// TIA Portal V18 export
ORGANIZATION_BLOCK "11-Bridge Movements"   // OB123, LAD, ProgramCycle
TITLE = Wheel
{ S7_Optimized_Access := 'TRUE' }
VERSION : 0.1
// stored: AutoNumber true, IsIECCheckEnabled false, SetENOAutomatically false
   VAR_INPUT
      Initial_Call : Bool;   // Initial call of this OB
      Remanence : Bool;   // =True, if remanent data are available
   END_VAR
   VAR_TEMP   // added for the SCL form of the ladder/FBD networks
      _w1 : Bool;
      _w2 : Bool;
      _w3 : Bool;
      _w4 : Bool;
   END_VAR
BEGIN

REGION Network 1: JoyStick MID
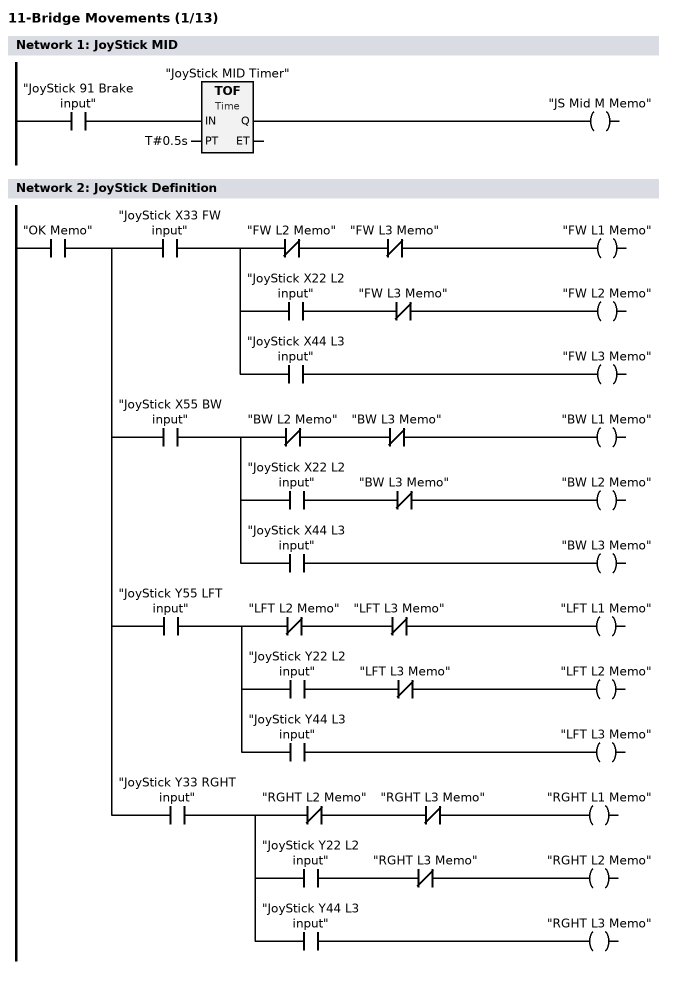
   RUNG wire#powerrail
      Contact( "JoyStick 91 Brake input" )
      { S7_Templates := "time_type := Time" } "JoyStick MID Timer".TOF(pt := T#0.5s, et =>)
      Coil( "JS Mid M Memo" )
   END_RUNG
   // the same network as SCL:
   "JoyStick MID Timer".TOF(IN := "JoyStick 91 Brake input", PT := T#0.5s);
   "JS Mid M Memo" := "JoyStick MID Timer".Q;
END_REGION

REGION Network 2: JoyStick Definition
   RUNG wire#powerrail
      Contact( "OK Memo" )
      wire#w1
      Contact( "JoyStick X33 FW input" )
      wire#w2
      I_Contact( "FW L2 Memo" )
      I_Contact( "FW L3 Memo" )
      Coil( "FW L1 Memo" )
   END_RUNG
   RUNG wire#w2
      Contact( "JoyStick X22 L2 input" )
      I_Contact( "FW L3 Memo" )
      Coil( "FW L2 Memo" )
   END_RUNG
   RUNG wire#w2
      Contact( "JoyStick X44 L3 input" )
      Coil( "FW L3 Memo" )
   END_RUNG
   RUNG wire#w1
      Contact( "JoyStick X55 BW input" )
      wire#w3
      I_Contact( "BW L2 Memo" )
      I_Contact( "BW L3 Memo" )
      Coil( "BW L1 Memo" )
   END_RUNG
   RUNG wire#w3
      Contact( "JoyStick X22 L2 input" )
      I_Contact( "BW L3 Memo" )
      Coil( "BW L2 Memo" )
   END_RUNG
   RUNG wire#w3
      Contact( "JoyStick X44 L3 input" )
      Coil( "BW L3 Memo" )
   END_RUNG
   RUNG wire#w1
      Contact( "JoyStick Y55 LFT input" )
      wire#w4
      I_Contact( "LFT L2 Memo" )
      I_Contact( "LFT L3 Memo" )
      Coil( "LFT L1 Memo" )
   END_RUNG
   RUNG wire#w4
      Contact( "JoyStick Y22 L2 input" )
      I_Contact( "LFT L3 Memo" )
      Coil( "LFT L2 Memo" )
   END_RUNG
   RUNG wire#w4
      Contact( "JoyStick Y44 L3 input" )
      Coil( "LFT L3 Memo" )
   END_RUNG
   RUNG wire#w1
      Contact( "JoyStick Y33 RGHT input" )
      wire#w5
      I_Contact( "RGHT L2 Memo" )
      I_Contact( "RGHT L3 Memo" )
      Coil( "RGHT L1 Memo" )
   END_RUNG
   RUNG wire#w5
      Contact( "JoyStick Y22 L2 input" )
      I_Contact( "RGHT L3 Memo" )
      Coil( "RGHT L2 Memo" )
   END_RUNG
   RUNG wire#w5
      Contact( "JoyStick Y44 L3 input" )
      Coil( "RGHT L3 Memo" )
   END_RUNG
   // the same network as SCL:
   #_w1 := "OK Memo" AND "JoyStick X33 FW input";
   "FW L1 Memo" := #_w1 AND NOT "FW L2 Memo" AND NOT "FW L3 Memo";
   "FW L2 Memo" := #_w1 AND "JoyStick X22 L2 input" AND NOT "FW L3 Memo";
   "FW L3 Memo" := #_w1 AND "JoyStick X44 L3 input";
   #_w2 := "OK Memo" AND "JoyStick X55 BW input";
   "BW L1 Memo" := #_w2 AND NOT "BW L2 Memo" AND NOT "BW L3 Memo";
   "BW L2 Memo" := #_w2 AND "JoyStick X22 L2 input" AND NOT "BW L3 Memo";
   "BW L3 Memo" := #_w2 AND "JoyStick X44 L3 input";
   #_w3 := "OK Memo" AND "JoyStick Y55 LFT input";
   "LFT L1 Memo" := #_w3 AND NOT "LFT L2 Memo" AND NOT "LFT L3 Memo";
   "LFT L2 Memo" := #_w3 AND "JoyStick Y22 L2 input" AND NOT "LFT L3 Memo";
   "LFT L3 Memo" := #_w3 AND "JoyStick Y44 L3 input";
   #_w4 := "OK Memo" AND "JoyStick Y33 RGHT input";
   "RGHT L1 Memo" := #_w4 AND NOT "RGHT L2 Memo" AND NOT "RGHT L3 Memo";
   "RGHT L2 Memo" := #_w4 AND "JoyStick Y22 L2 input" AND NOT "RGHT L3 Memo";
   "RGHT L3 Memo" := #_w4 AND "JoyStick Y44 L3 input";
END_REGION

REGION Network 3: JoyStick Cross Definition
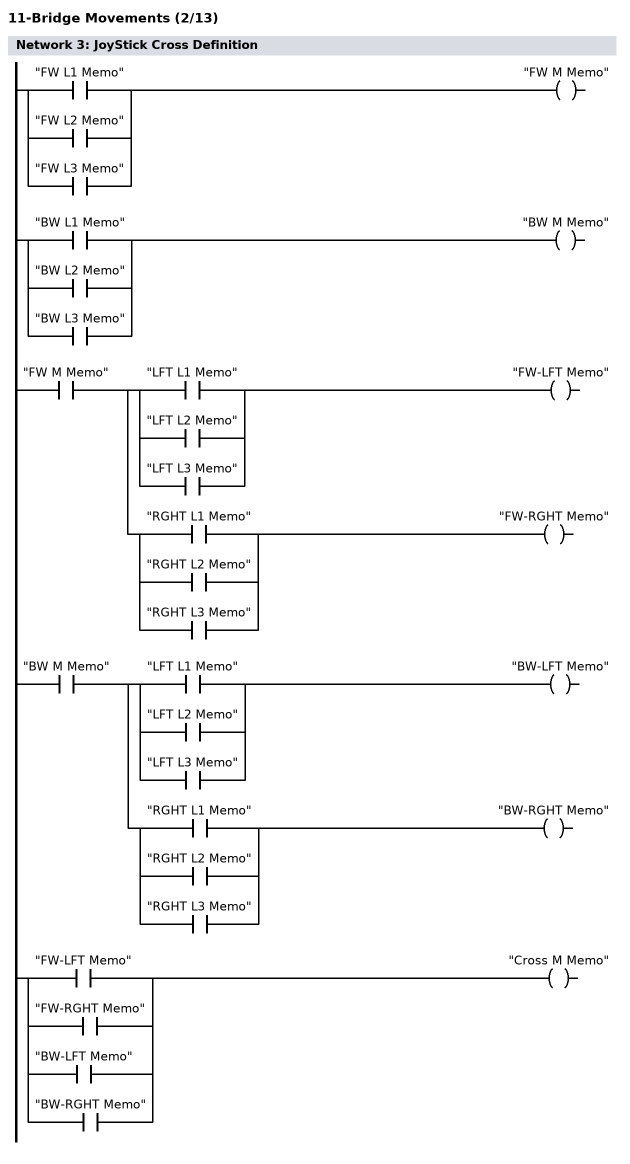
   RUNG wire#powerrail
      Contact( "FW L1 Memo" )
      wire#w1
      Coil( "FW M Memo" )
   END_RUNG
   RUNG wire#powerrail
      Contact( "FW L2 Memo" )
   END_RUNG wire#w1
   RUNG wire#powerrail
      Contact( "FW L3 Memo" )
   END_RUNG wire#w1
   RUNG wire#powerrail
      Contact( "BW L1 Memo" )
      wire#w2
      Coil( "BW M Memo" )
   END_RUNG
   RUNG wire#powerrail
      Contact( "BW L2 Memo" )
   END_RUNG wire#w2
   RUNG wire#powerrail
      Contact( "BW L3 Memo" )
   END_RUNG wire#w2
   RUNG wire#powerrail
      Contact( "FW M Memo" )
      wire#w3
      Contact( "LFT L1 Memo" )
      wire#w4
      Coil( "FW-LFT Memo" )
   END_RUNG
   RUNG wire#w3
      Contact( "LFT L2 Memo" )
   END_RUNG wire#w4
   RUNG wire#w3
      Contact( "LFT L3 Memo" )
   END_RUNG wire#w4
   RUNG wire#w3
      Contact( "RGHT L1 Memo" )
      wire#w5
      Coil( "FW-RGHT Memo" )
   END_RUNG
   RUNG wire#w3
      Contact( "RGHT L2 Memo" )
   END_RUNG wire#w5
   RUNG wire#w3
      Contact( "RGHT L3 Memo" )
   END_RUNG wire#w5
   RUNG wire#powerrail
      Contact( "BW M Memo" )
      wire#w6
      Contact( "LFT L1 Memo" )
      wire#w7
      Coil( "BW-LFT Memo" )
   END_RUNG
   RUNG wire#w6
      Contact( "LFT L2 Memo" )
   END_RUNG wire#w7
   RUNG wire#w6
      Contact( "LFT L3 Memo" )
   END_RUNG wire#w7
   RUNG wire#w6
      Contact( "RGHT L1 Memo" )
      wire#w8
      Coil( "BW-RGHT Memo" )
   END_RUNG
   RUNG wire#w6
      Contact( "RGHT L2 Memo" )
   END_RUNG wire#w8
   RUNG wire#w6
      Contact( "RGHT L3 Memo" )
   END_RUNG wire#w8
   RUNG wire#powerrail
      Contact( "FW-LFT Memo" )
      wire#w9
      Coil( "Cross M Memo" )
   END_RUNG
   RUNG wire#powerrail
      Contact( "FW-RGHT Memo" )
   END_RUNG wire#w9
   RUNG wire#powerrail
      Contact( "BW-LFT Memo" )
   END_RUNG wire#w9
   RUNG wire#powerrail
      Contact( "BW-RGHT Memo" )
   END_RUNG wire#w9
   // the same network as SCL:
   "FW M Memo" := "FW L1 Memo" OR "FW L2 Memo" OR "FW L3 Memo";
   "BW M Memo" := "BW L1 Memo" OR "BW L2 Memo" OR "BW L3 Memo";
   "FW-LFT Memo" := "FW M Memo" AND ("LFT L1 Memo" OR "LFT L2 Memo" OR "LFT L3 Memo");
   "FW-RGHT Memo" := "FW M Memo" AND ("RGHT L1 Memo" OR "RGHT L2 Memo" OR "RGHT L3 Memo");
   "BW-LFT Memo" := "BW M Memo" AND ("LFT L1 Memo" OR "LFT L2 Memo" OR "LFT L3 Memo");
   "BW-RGHT Memo" := "BW M Memo" AND ("RGHT L1 Memo" OR "RGHT L2 Memo" OR "RGHT L3 Memo");
   "Cross M Memo" := "FW-LFT Memo" OR "FW-RGHT Memo" OR "BW-LFT Memo" OR "BW-RGHT Memo";
END_REGION

REGION Network 4: Speed Settings
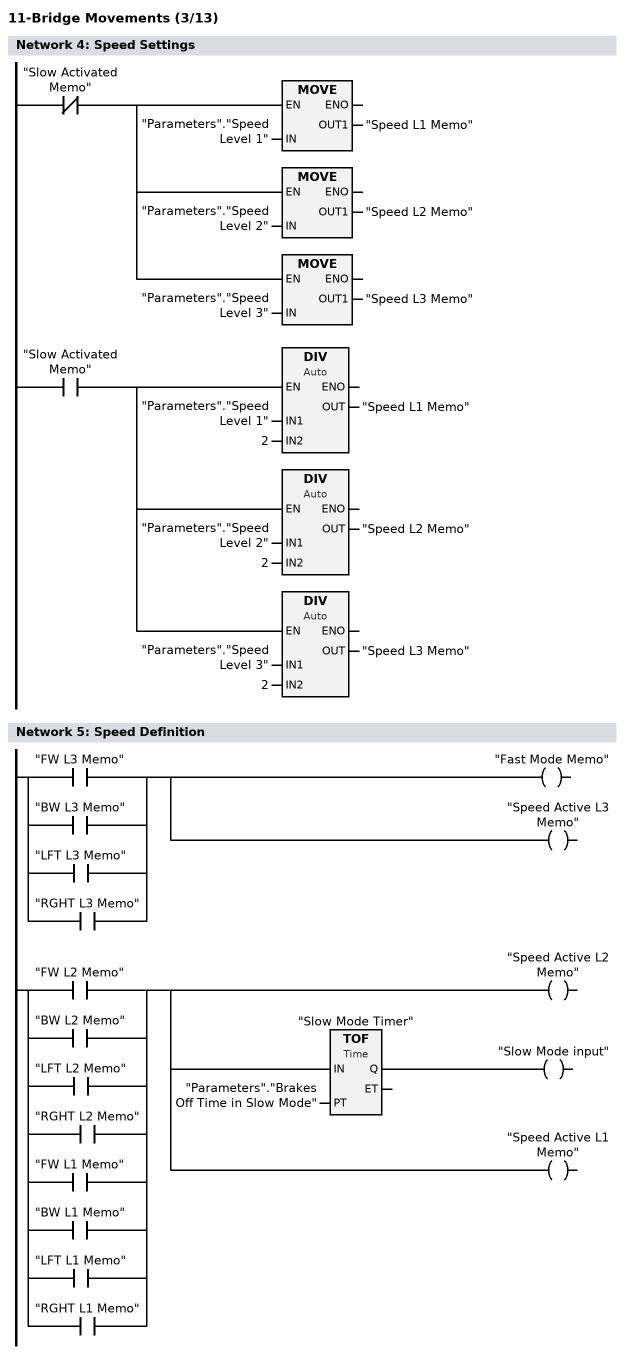
   RUNG wire#powerrail
      I_Contact( "Slow Activated Memo" )
      wire#w1
      Move(in := "Parameters"."Speed Level 1", out1 => "Speed L1 Memo")
   END_RUNG
   RUNG wire#w1
      Move(in := "Parameters"."Speed Level 2", out1 => "Speed L2 Memo")
   END_RUNG
   RUNG wire#w1
      Move(in := "Parameters"."Speed Level 3", out1 => "Speed L3 Memo")
   END_RUNG
   RUNG wire#powerrail
      Contact( "Slow Activated Memo" )
      wire#w2
      Div(in1 := "Parameters"."Speed Level 1", in2 := 2, out => "Speed L1 Memo")
   END_RUNG
   RUNG wire#w2
      Div(in1 := "Parameters"."Speed Level 2", in2 := 2, out => "Speed L2 Memo")
   END_RUNG
   RUNG wire#w2
      Div(in1 := "Parameters"."Speed Level 3", in2 := 2, out => "Speed L3 Memo")
   END_RUNG
   // the same network as SCL:
   IF NOT "Slow Activated Memo" THEN
       "Speed L1 Memo" := "Parameters"."Speed Level 1";
       "Speed L2 Memo" := "Parameters"."Speed Level 2";
       "Speed L3 Memo" := "Parameters"."Speed Level 3";
   END_IF;
   IF "Slow Activated Memo" THEN
       "Speed L1 Memo" := "Parameters"."Speed Level 1" / 2;
       "Speed L2 Memo" := "Parameters"."Speed Level 2" / 2;
       "Speed L3 Memo" := "Parameters"."Speed Level 3" / 2;
   END_IF;
END_REGION

REGION Network 5: Speed Definition
   RUNG wire#powerrail
      Contact( "FW L3 Memo" )
      wire#w1
      Coil( "Fast Mode Memo" )
   END_RUNG
   RUNG wire#powerrail
      Contact( "BW L3 Memo" )
   END_RUNG wire#w1
   RUNG wire#powerrail
      Contact( "LFT L3 Memo" )
   END_RUNG wire#w1
   RUNG wire#powerrail
      Contact( "RGHT L3 Memo" )
   END_RUNG wire#w1
   RUNG wire#w1
      Coil( "Speed Active L3 Memo" )
   END_RUNG
   RUNG wire#powerrail
      Contact( "FW L2 Memo" )
      wire#w2
      Coil( "Speed Active L2 Memo" )
   END_RUNG
   RUNG wire#powerrail
      Contact( "BW L2 Memo" )
   END_RUNG wire#w2
   RUNG wire#powerrail
      Contact( "LFT L2 Memo" )
   END_RUNG wire#w2
   RUNG wire#powerrail
      Contact( "RGHT L2 Memo" )
   END_RUNG wire#w2
   RUNG wire#powerrail
      Contact( "FW L1 Memo" )
   END_RUNG wire#w2
   RUNG wire#powerrail
      Contact( "BW L1 Memo" )
   END_RUNG wire#w2
   RUNG wire#powerrail
      Contact( "LFT L1 Memo" )
   END_RUNG wire#w2
   RUNG wire#powerrail
      Contact( "RGHT L1 Memo" )
   END_RUNG wire#w2
   RUNG wire#w2
      { S7_Templates := "time_type := Time" } "Slow Mode Timer".TOF(pt := "Parameters"."Brakes Off Time in Slow Mode", et =>)
      Coil( "Slow Mode input" )
   END_RUNG
   RUNG wire#w2
      Coil( "Speed Active L1 Memo" )
   END_RUNG
   // the same network as SCL:
   "Fast Mode Memo" := "FW L3 Memo" OR "BW L3 Memo" OR "LFT L3 Memo" OR "RGHT L3 Memo";
   "Speed Active L3 Memo" := "Fast Mode Memo";
   "Speed Active L2 Memo" := "FW L2 Memo" OR "BW L2 Memo" OR "LFT L2 Memo" OR "RGHT L2 Memo" OR "FW L1 Memo" OR "BW L1 Memo" OR "LFT L1 Memo" OR "RGHT L1 Memo";
   "Slow Mode Timer".TOF(IN := "Speed Active L2 Memo", PT := "Parameters"."Brakes Off Time in Slow Mode");
   "Slow Mode input" := "Slow Mode Timer".Q;
   "Speed Active L1 Memo" := "Speed Active L2 Memo";
END_REGION

REGION Network 6: Slow Activated
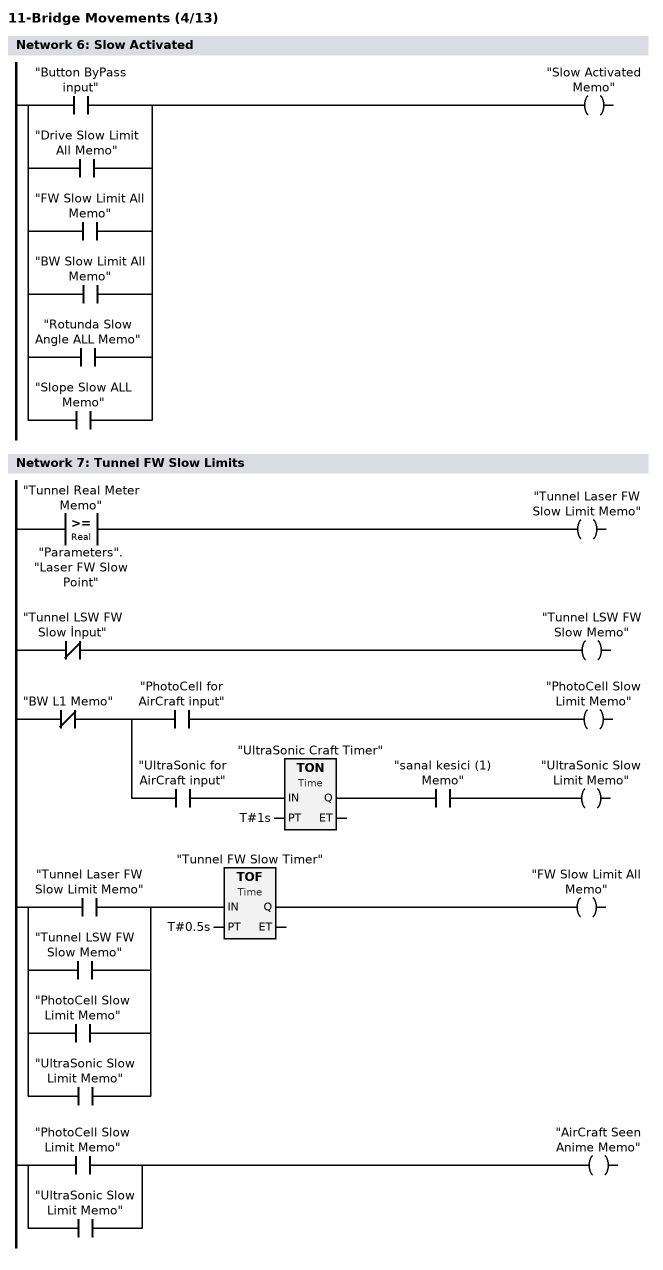
   RUNG wire#powerrail
      Contact( "Button ByPass input" )
      wire#w1
      Coil( "Slow Activated Memo" )
   END_RUNG
   RUNG wire#powerrail
      Contact( "Drive Slow Limit All Memo" )
   END_RUNG wire#w1
   RUNG wire#powerrail
      Contact( "FW Slow Limit All Memo" )
   END_RUNG wire#w1
   RUNG wire#powerrail
      Contact( "BW Slow Limit All Memo" )
   END_RUNG wire#w1
   RUNG wire#powerrail
      Contact( "Rotunda Slow Angle ALL Memo" )
   END_RUNG wire#w1
   RUNG wire#powerrail
      Contact( "Slope Slow ALL Memo" )
   END_RUNG wire#w1
   // the same network as SCL:
   "Slow Activated Memo" := "Button ByPass input" OR "Drive Slow Limit All Memo" OR "FW Slow Limit All Memo" OR "BW Slow Limit All Memo" OR "Rotunda Slow Angle ALL Memo" OR "Slope Slow ALL Memo";
END_REGION

REGION Network 7: Tunnel FW Slow Limits
   RUNG wire#powerrail
      { S7_Templates := "SrcType := Real" } GE_Contact(in1 := "Tunnel Real Meter Memo", in2 := "Parameters"."Laser FW Slow Point")
      Coil( "Tunnel Laser FW Slow Limit Memo" )
   END_RUNG
   RUNG wire#powerrail
      I_Contact( "Tunnel LSW FW Slow İnput" )
      Coil( "Tunnel LSW FW Slow Memo" )
   END_RUNG
   RUNG wire#powerrail
      I_Contact( "BW L1 Memo" )
      wire#w1
      Contact( "PhotoCell for AirCraft input" )
      Coil( "PhotoCell Slow Limit Memo" )
   END_RUNG
   RUNG wire#w1
      Contact( "UltraSonic for AirCraft input" )
      { S7_Templates := "time_type := Time" } "UltraSonic Craft Timer".TON(pt := T#1s, et =>)
      Contact( "sanal kesici (1) Memo" )
      Coil( "UltraSonic Slow Limit Memo" )
   END_RUNG
   RUNG wire#powerrail
      Contact( "Tunnel Laser FW Slow Limit Memo" )
      wire#w2
      { S7_Templates := "time_type := Time" } "Tunnel FW Slow Timer".TOF(pt := T#0.5s, et =>)
      Coil( "FW Slow Limit All Memo" )
   END_RUNG
   RUNG wire#powerrail
      Contact( "Tunnel LSW FW Slow Memo" )
   END_RUNG wire#w2
   RUNG wire#powerrail
      Contact( "PhotoCell Slow Limit Memo" )
   END_RUNG wire#w2
   RUNG wire#powerrail
      Contact( "UltraSonic Slow Limit Memo" )
   END_RUNG wire#w2
   RUNG wire#powerrail
      Contact( "PhotoCell Slow Limit Memo" )
      wire#w3
      Coil( "AirCraft Seen Anime Memo" )
   END_RUNG
   RUNG wire#powerrail
      Contact( "UltraSonic Slow Limit Memo" )
   END_RUNG wire#w3
   // the same network as SCL:
   "Tunnel Laser FW Slow Limit Memo" := "Tunnel Real Meter Memo" >= "Parameters"."Laser FW Slow Point";
   "Tunnel LSW FW Slow Memo" := NOT "Tunnel LSW FW Slow İnput";
   "PhotoCell Slow Limit Memo" := NOT "BW L1 Memo" AND "PhotoCell for AirCraft input";
   "UltraSonic Craft Timer".TON(IN := NOT "BW L1 Memo" AND "UltraSonic for AirCraft input", PT := T#1s);
   "UltraSonic Slow Limit Memo" := "UltraSonic Craft Timer".Q AND "sanal kesici (1) Memo";
   "Tunnel FW Slow Timer".TOF(IN := "Tunnel Laser FW Slow Limit Memo" OR "Tunnel LSW FW Slow Memo" OR "PhotoCell Slow Limit Memo" OR "UltraSonic Slow Limit Memo",
                           PT := T#0.5s);
   "FW Slow Limit All Memo" := "Tunnel FW Slow Timer".Q;
   "AirCraft Seen Anime Memo" := "PhotoCell Slow Limit Memo" OR "UltraSonic Slow Limit Memo";
END_REGION

REGION Network 8: Tunnel BW Slow Limits
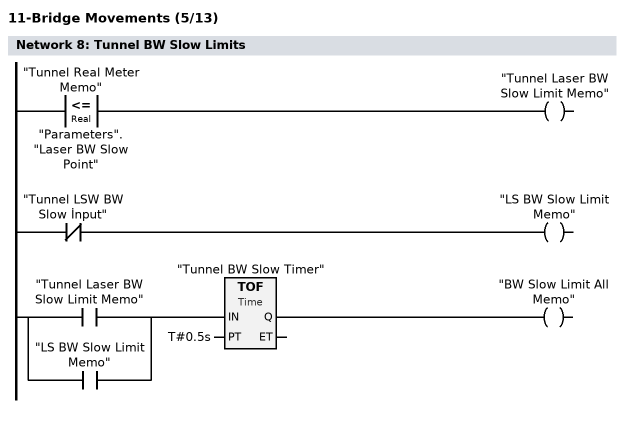
   RUNG wire#powerrail
      { S7_Templates := "SrcType := Real" } LE_Contact(in1 := "Tunnel Real Meter Memo", in2 := "Parameters"."Laser BW Slow Point")
      Coil( "Tunnel Laser BW Slow Limit Memo" )
   END_RUNG
   RUNG wire#powerrail
      I_Contact( "Tunnel LSW BW Slow İnput" )
      Coil( "LS BW Slow Limit Memo" )
   END_RUNG
   RUNG wire#powerrail
      Contact( "Tunnel Laser BW Slow Limit Memo" )
      wire#w1
      { S7_Templates := "time_type := Time" } "Tunnel BW Slow Timer".TOF(pt := T#0.5s, et =>)
      Coil( "BW Slow Limit All Memo" )
   END_RUNG
   RUNG wire#powerrail
      Contact( "LS BW Slow Limit Memo" )
   END_RUNG wire#w1
   // the same network as SCL:
   "Tunnel Laser BW Slow Limit Memo" := "Tunnel Real Meter Memo" <= "Parameters"."Laser BW Slow Point";
   "LS BW Slow Limit Memo" := NOT "Tunnel LSW BW Slow İnput";
   "Tunnel BW Slow Timer".TOF(IN := "Tunnel Laser BW Slow Limit Memo" OR "LS BW Slow Limit Memo", PT := T#0.5s);
   "BW Slow Limit All Memo" := "Tunnel BW Slow Timer".Q;
END_REGION

REGION Network 9: Tunnel FW Stop Limits
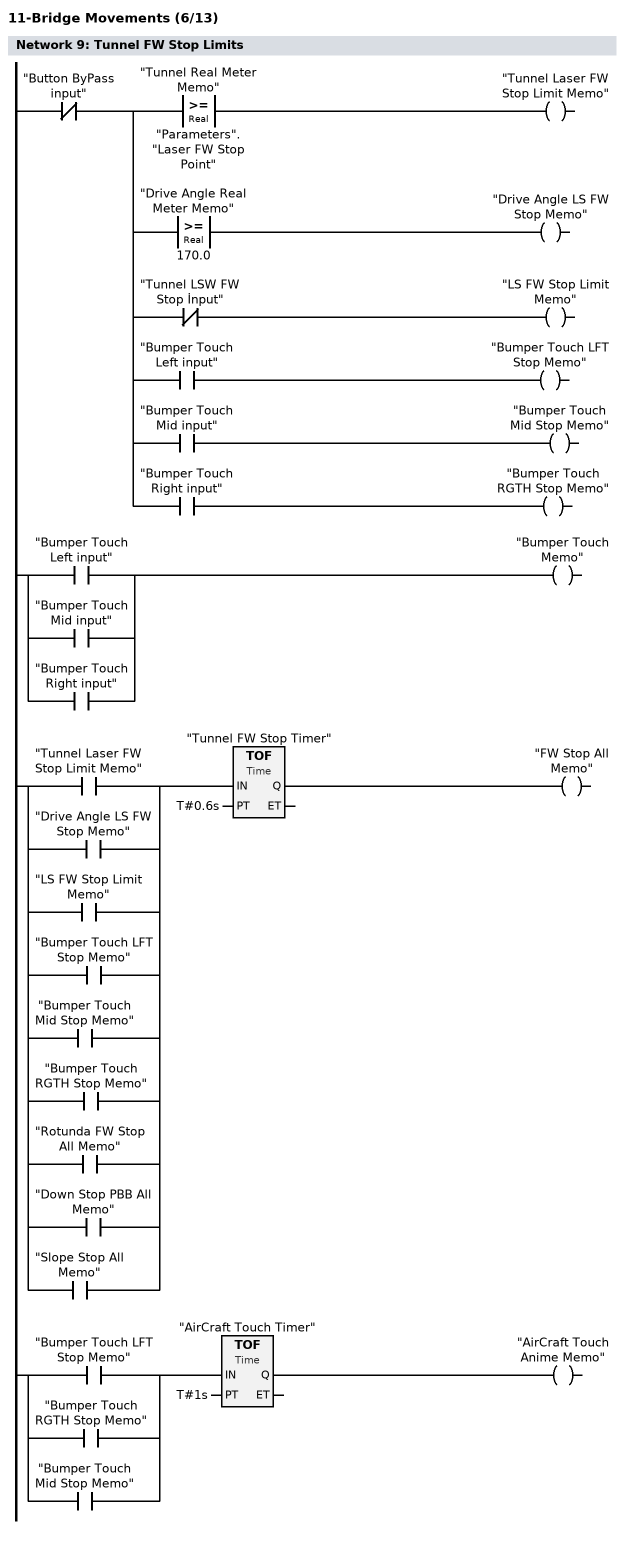
   RUNG wire#powerrail
      I_Contact( "Button ByPass input" )
      wire#w1
      { S7_Templates := "SrcType := Real" } GE_Contact(in1 := "Tunnel Real Meter Memo", in2 := "Parameters"."Laser FW Stop Point")
      Coil( "Tunnel Laser FW Stop Limit Memo" )
   END_RUNG
   RUNG wire#w1
      { S7_Templates := "SrcType := Real" } GE_Contact(in1 := "Drive Angle Real Meter Memo", in2 := 170.0)
      Coil( "Drive Angle LS FW Stop Memo" )
   END_RUNG
   RUNG wire#w1
      I_Contact( "Tunnel LSW FW Stop İnput" )
      Coil( "LS FW Stop Limit Memo" )
   END_RUNG
   RUNG wire#w1
      Contact( "Bumper Touch Left input" )
      Coil( "Bumper Touch LFT Stop Memo" )
   END_RUNG
   RUNG wire#w1
      Contact( "Bumper Touch Mid input" )
      Coil( "Bumper Touch Mid Stop Memo" )
   END_RUNG
   RUNG wire#w1
      Contact( "Bumper Touch Right input" )
      Coil( "Bumper Touch RGTH Stop Memo" )
   END_RUNG
   RUNG wire#powerrail
      Contact( "Bumper Touch Left input" )
      wire#w2
      Coil( "Bumper Touch Memo" )
   END_RUNG
   RUNG wire#powerrail
      Contact( "Bumper Touch Mid input" )
   END_RUNG wire#w2
   RUNG wire#powerrail
      Contact( "Bumper Touch Right input" )
   END_RUNG wire#w2
   RUNG wire#powerrail
      Contact( "Tunnel Laser FW Stop Limit Memo" )
      wire#w3
      { S7_Templates := "time_type := Time" } "Tunnel FW Stop Timer".TOF(pt := T#0.6s, et =>)
      Coil( "FW Stop All Memo" )
   END_RUNG
   RUNG wire#powerrail
      Contact( "Drive Angle LS FW Stop Memo" )
   END_RUNG wire#w3
   RUNG wire#powerrail
      Contact( "LS FW Stop Limit Memo" )
   END_RUNG wire#w3
   RUNG wire#powerrail
      Contact( "Bumper Touch LFT Stop Memo" )
   END_RUNG wire#w3
   RUNG wire#powerrail
      Contact( "Bumper Touch Mid Stop Memo" )
   END_RUNG wire#w3
   RUNG wire#powerrail
      Contact( "Bumper Touch RGTH Stop Memo" )
   END_RUNG wire#w3
   RUNG wire#powerrail
      Contact( "Rotunda FW Stop All Memo" )
   END_RUNG wire#w3
   RUNG wire#powerrail
      Contact( "Down Stop PBB All Memo" )
   END_RUNG wire#w3
   RUNG wire#powerrail
      Contact( "Slope Stop All Memo" )
   END_RUNG wire#w3
   RUNG wire#powerrail
      Contact( "Bumper Touch LFT Stop Memo" )
      wire#w4
      { S7_Templates := "time_type := Time" } "AirCraft Touch Timer".TOF(pt := T#1s, et =>)
      Coil( "AirCraft Touch Anime Memo" )
   END_RUNG
   RUNG wire#powerrail
      Contact( "Bumper Touch RGTH Stop Memo" )
   END_RUNG wire#w4
   RUNG wire#powerrail
      Contact( "Bumper Touch Mid Stop Memo" )
   END_RUNG wire#w4
   // the same network as SCL:
   #_w1 := NOT "Button ByPass input";
   "Tunnel Laser FW Stop Limit Memo" := #_w1 AND ("Tunnel Real Meter Memo" >= "Parameters"."Laser FW Stop Point");
   "Drive Angle LS FW Stop Memo" := #_w1 AND ("Drive Angle Real Meter Memo" >= 170.0);
   "LS FW Stop Limit Memo" := #_w1 AND NOT "Tunnel LSW FW Stop İnput";
   "Bumper Touch LFT Stop Memo" := #_w1 AND "Bumper Touch Left input";
   "Bumper Touch Mid Stop Memo" := #_w1 AND "Bumper Touch Mid input";
   "Bumper Touch RGTH Stop Memo" := #_w1 AND "Bumper Touch Right input";
   "Bumper Touch Memo" := "Bumper Touch Left input" OR "Bumper Touch Mid input" OR "Bumper Touch Right input";
   "Tunnel FW Stop Timer".TOF(IN := "Tunnel Laser FW Stop Limit Memo" OR "Drive Angle LS FW Stop Memo" OR "LS FW Stop Limit Memo" OR "Bumper Touch LFT Stop Memo" OR "Bumper Touch Mid Stop Memo" OR "Bumper Touch RGTH Stop Memo" OR "Rotunda FW Stop All Memo" OR "Down Stop PBB All Memo" OR "Slope Stop All Memo",
                           PT := T#0.6s);
   "FW Stop All Memo" := "Tunnel FW Stop Timer".Q;
   "AirCraft Touch Timer".TOF(IN := "Bumper Touch LFT Stop Memo" OR "Bumper Touch RGTH Stop Memo" OR "Bumper Touch Mid Stop Memo",
                           PT := T#1s);
   "AirCraft Touch Anime Memo" := "AirCraft Touch Timer".Q;
END_REGION

REGION Network 10: Tunnel BW Stop Limits
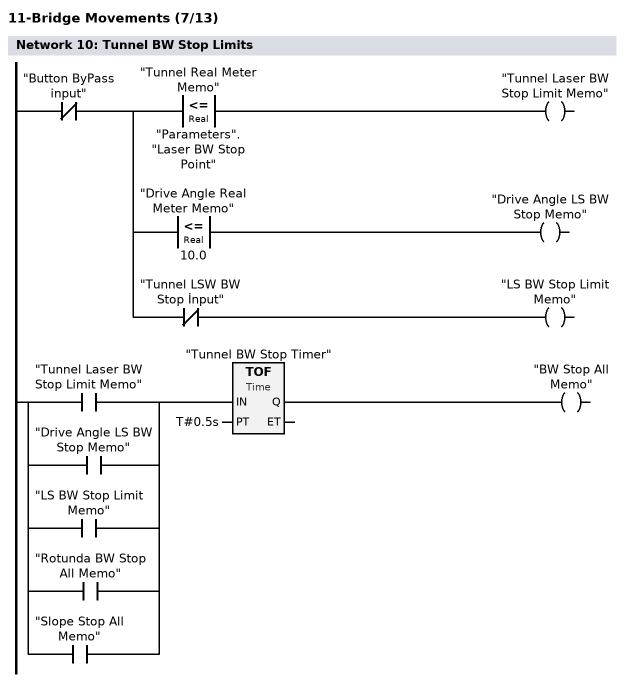
   RUNG wire#powerrail
      I_Contact( "Button ByPass input" )
      wire#w1
      { S7_Templates := "SrcType := Real" } LE_Contact(in1 := "Tunnel Real Meter Memo", in2 := "Parameters"."Laser BW Stop Point")
      Coil( "Tunnel Laser BW Stop Limit Memo" )
   END_RUNG
   RUNG wire#w1
      { S7_Templates := "SrcType := Real" } LE_Contact(in1 := "Drive Angle Real Meter Memo", in2 := 10.0)
      Coil( "Drive Angle LS BW Stop Memo" )
   END_RUNG
   RUNG wire#w1
      I_Contact( "Tunnel LSW BW Stop İnput" )
      Coil( "LS BW Stop Limit Memo" )
   END_RUNG
   RUNG wire#powerrail
      Contact( "Tunnel Laser BW Stop Limit Memo" )
      wire#w2
      { S7_Templates := "time_type := Time" } "Tunnel BW Stop Timer".TOF(pt := T#0.5s, et =>)
      Coil( "BW Stop All Memo" )
   END_RUNG
   RUNG wire#powerrail
      Contact( "Drive Angle LS BW Stop Memo" )
   END_RUNG wire#w2
   RUNG wire#powerrail
      Contact( "LS BW Stop Limit Memo" )
   END_RUNG wire#w2
   RUNG wire#powerrail
      Contact( "Rotunda BW Stop All Memo" )
   END_RUNG wire#w2
   RUNG wire#powerrail
      Contact( "Slope Stop All Memo" )
   END_RUNG wire#w2
   // the same network as SCL:
   #_w1 := NOT "Button ByPass input";
   "Tunnel Laser BW Stop Limit Memo" := #_w1 AND ("Tunnel Real Meter Memo" <= "Parameters"."Laser BW Stop Point");
   "Drive Angle LS BW Stop Memo" := #_w1 AND ("Drive Angle Real Meter Memo" <= 10.0);
   "LS BW Stop Limit Memo" := #_w1 AND NOT "Tunnel LSW BW Stop İnput";
   "Tunnel BW Stop Timer".TOF(IN := "Tunnel Laser BW Stop Limit Memo" OR "Drive Angle LS BW Stop Memo" OR "LS BW Stop Limit Memo" OR "Rotunda BW Stop All Memo" OR "Slope Stop All Memo",
                           PT := T#0.5s);
   "BW Stop All Memo" := "Tunnel BW Stop Timer".Q;
END_REGION

REGION Network 11: Tunnel FW
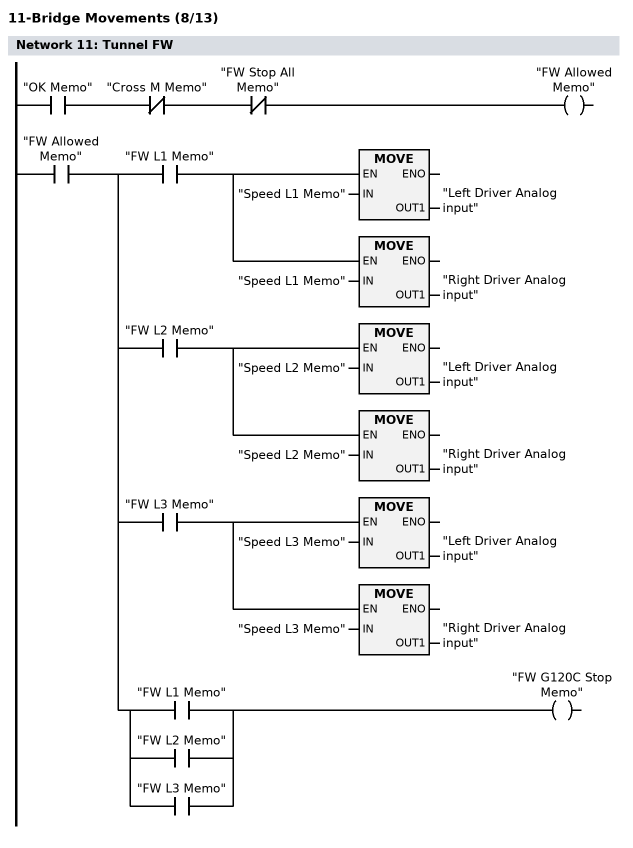
   RUNG wire#powerrail
      Contact( "OK Memo" )
      I_Contact( "Cross M Memo" )
      I_Contact( "FW Stop All Memo" )
      Coil( "FW Allowed Memo" )
   END_RUNG
   RUNG wire#powerrail
      Contact( "FW Allowed Memo" )
      wire#w1
      Contact( "FW L1 Memo" )
      wire#w2
      Move(in := "Speed L1 Memo", out1 => "Left Driver Analog input")
   END_RUNG
   RUNG wire#w2
      Move(in := "Speed L1 Memo", out1 => "Right Driver Analog input")
   END_RUNG
   RUNG wire#w1
      Contact( "FW L2 Memo" )
      wire#w3
      Move(in := "Speed L2 Memo", out1 => "Left Driver Analog input")
   END_RUNG
   RUNG wire#w3
      Move(in := "Speed L2 Memo", out1 => "Right Driver Analog input")
   END_RUNG
   RUNG wire#w1
      Contact( "FW L3 Memo" )
      wire#w4
      Move(in := "Speed L3 Memo", out1 => "Left Driver Analog input")
   END_RUNG
   RUNG wire#w4
      Move(in := "Speed L3 Memo", out1 => "Right Driver Analog input")
   END_RUNG
   RUNG wire#w1
      Contact( "FW L1 Memo" )
      wire#w5
      Coil( "FW G120C Stop Memo" )
   END_RUNG
   RUNG wire#w1
      Contact( "FW L2 Memo" )
   END_RUNG wire#w5
   RUNG wire#w1
      Contact( "FW L3 Memo" )
   END_RUNG wire#w5
   // the same network as SCL:
   "FW Allowed Memo" := "OK Memo" AND NOT "Cross M Memo" AND NOT "FW Stop All Memo";
   IF "FW Allowed Memo" AND "FW L1 Memo" THEN
       "Left Driver Analog input" := "Speed L1 Memo";
       "Right Driver Analog input" := "Speed L1 Memo";
   END_IF;
   IF "FW Allowed Memo" AND "FW L2 Memo" THEN
       "Left Driver Analog input" := "Speed L2 Memo";
       "Right Driver Analog input" := "Speed L2 Memo";
   END_IF;
   IF "FW Allowed Memo" AND "FW L3 Memo" THEN
       "Left Driver Analog input" := "Speed L3 Memo";
       "Right Driver Analog input" := "Speed L3 Memo";
   END_IF;
   "FW G120C Stop Memo" := "FW Allowed Memo" AND ("FW L1 Memo" OR "FW L2 Memo" OR "FW L3 Memo");
END_REGION

REGION Network 12: Tunnel BW
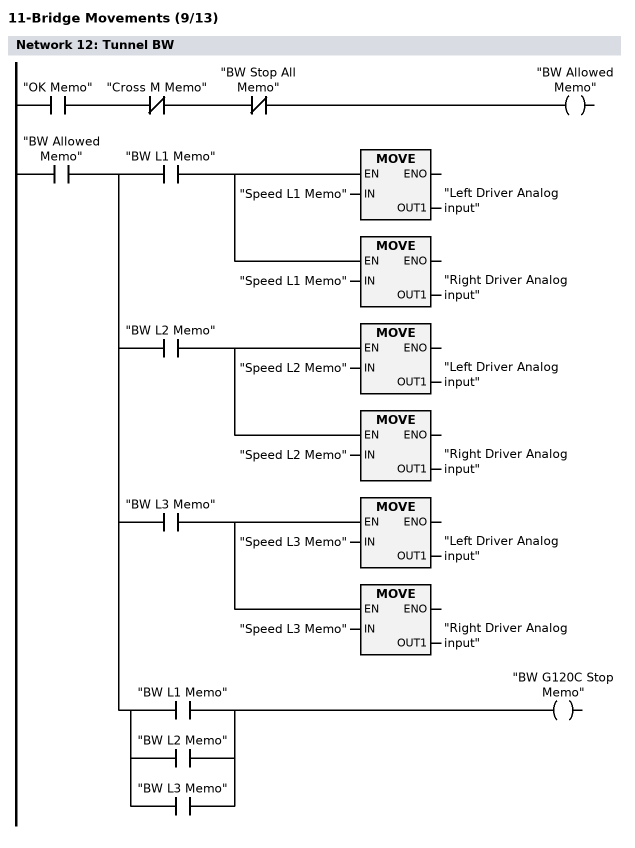
   RUNG wire#powerrail
      Contact( "OK Memo" )
      I_Contact( "Cross M Memo" )
      I_Contact( "BW Stop All Memo" )
      Coil( "BW Allowed Memo" )
   END_RUNG
   RUNG wire#powerrail
      Contact( "BW Allowed Memo" )
      wire#w1
      Contact( "BW L1 Memo" )
      wire#w2
      Move(in := "Speed L1 Memo", out1 => "Left Driver Analog input")
   END_RUNG
   RUNG wire#w2
      Move(in := "Speed L1 Memo", out1 => "Right Driver Analog input")
   END_RUNG
   RUNG wire#w1
      Contact( "BW L2 Memo" )
      wire#w3
      Move(in := "Speed L2 Memo", out1 => "Left Driver Analog input")
   END_RUNG
   RUNG wire#w3
      Move(in := "Speed L2 Memo", out1 => "Right Driver Analog input")
   END_RUNG
   RUNG wire#w1
      Contact( "BW L3 Memo" )
      wire#w4
      Move(in := "Speed L3 Memo", out1 => "Left Driver Analog input")
   END_RUNG
   RUNG wire#w4
      Move(in := "Speed L3 Memo", out1 => "Right Driver Analog input")
   END_RUNG
   RUNG wire#w1
      Contact( "BW L1 Memo" )
      wire#w5
      Coil( "BW G120C Stop Memo" )
   END_RUNG
   RUNG wire#w1
      Contact( "BW L2 Memo" )
   END_RUNG wire#w5
   RUNG wire#w1
      Contact( "BW L3 Memo" )
   END_RUNG wire#w5
   // the same network as SCL:
   "BW Allowed Memo" := "OK Memo" AND NOT "Cross M Memo" AND NOT "BW Stop All Memo";
   IF "BW Allowed Memo" AND "BW L1 Memo" THEN
       "Left Driver Analog input" := "Speed L1 Memo";
       "Right Driver Analog input" := "Speed L1 Memo";
   END_IF;
   IF "BW Allowed Memo" AND "BW L2 Memo" THEN
       "Left Driver Analog input" := "Speed L2 Memo";
       "Right Driver Analog input" := "Speed L2 Memo";
   END_IF;
   IF "BW Allowed Memo" AND "BW L3 Memo" THEN
       "Left Driver Analog input" := "Speed L3 Memo";
       "Right Driver Analog input" := "Speed L3 Memo";
   END_IF;
   "BW G120C Stop Memo" := "BW Allowed Memo" AND ("BW L1 Memo" OR "BW L2 Memo" OR "BW L3 Memo");
END_REGION

REGION Network 13: Tunnel LFT
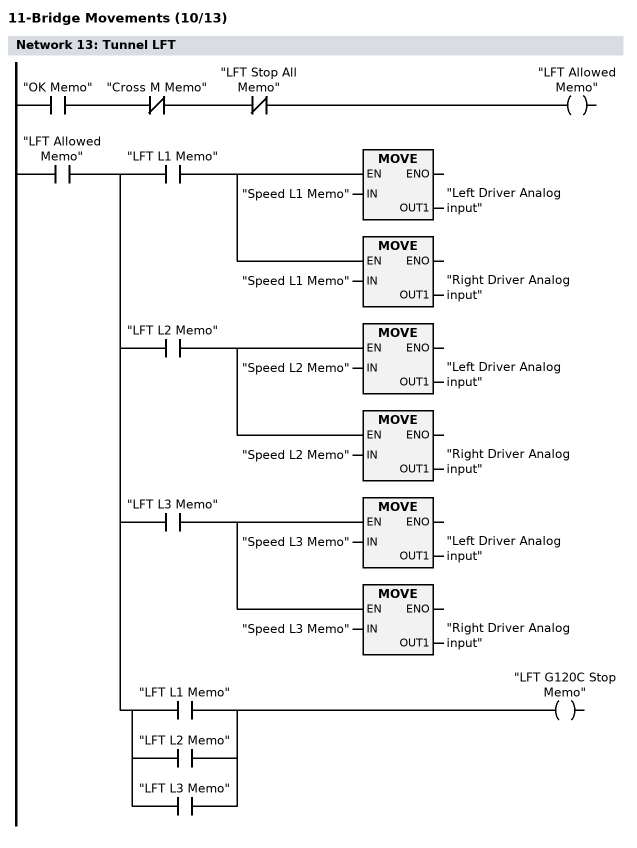
   RUNG wire#powerrail
      Contact( "OK Memo" )
      I_Contact( "Cross M Memo" )
      I_Contact( "LFT Stop All Memo" )
      Coil( "LFT Allowed Memo" )
   END_RUNG
   RUNG wire#powerrail
      Contact( "LFT Allowed Memo" )
      wire#w1
      Contact( "LFT L1 Memo" )
      wire#w2
      Move(in := "Speed L1 Memo", out1 => "Left Driver Analog input")
   END_RUNG
   RUNG wire#w2
      Move(in := "Speed L1 Memo", out1 => "Right Driver Analog input")
   END_RUNG
   RUNG wire#w1
      Contact( "LFT L2 Memo" )
      wire#w3
      Move(in := "Speed L2 Memo", out1 => "Left Driver Analog input")
   END_RUNG
   RUNG wire#w3
      Move(in := "Speed L2 Memo", out1 => "Right Driver Analog input")
   END_RUNG
   RUNG wire#w1
      Contact( "LFT L3 Memo" )
      wire#w4
      Move(in := "Speed L3 Memo", out1 => "Left Driver Analog input")
   END_RUNG
   RUNG wire#w4
      Move(in := "Speed L3 Memo", out1 => "Right Driver Analog input")
   END_RUNG
   RUNG wire#w1
      Contact( "LFT L1 Memo" )
      wire#w5
      Coil( "LFT G120C Stop Memo" )
   END_RUNG
   RUNG wire#w1
      Contact( "LFT L2 Memo" )
   END_RUNG wire#w5
   RUNG wire#w1
      Contact( "LFT L3 Memo" )
   END_RUNG wire#w5
   // the same network as SCL:
   "LFT Allowed Memo" := "OK Memo" AND NOT "Cross M Memo" AND NOT "LFT Stop All Memo";
   IF "LFT Allowed Memo" AND "LFT L1 Memo" THEN
       "Left Driver Analog input" := "Speed L1 Memo";
       "Right Driver Analog input" := "Speed L1 Memo";
   END_IF;
   IF "LFT Allowed Memo" AND "LFT L2 Memo" THEN
       "Left Driver Analog input" := "Speed L2 Memo";
       "Right Driver Analog input" := "Speed L2 Memo";
   END_IF;
   IF "LFT Allowed Memo" AND "LFT L3 Memo" THEN
       "Left Driver Analog input" := "Speed L3 Memo";
       "Right Driver Analog input" := "Speed L3 Memo";
   END_IF;
   "LFT G120C Stop Memo" := "LFT Allowed Memo" AND ("LFT L1 Memo" OR "LFT L2 Memo" OR "LFT L3 Memo");
END_REGION

REGION Network 14: Tunnel RGHT
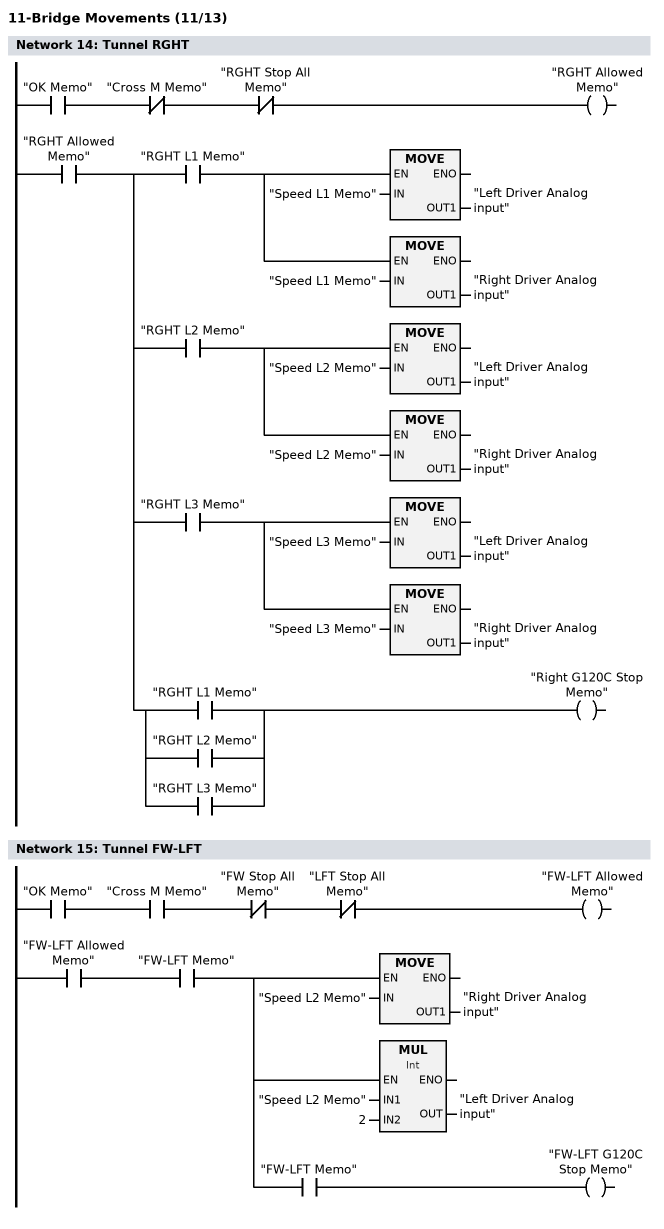
   RUNG wire#powerrail
      Contact( "OK Memo" )
      I_Contact( "Cross M Memo" )
      I_Contact( "RGHT Stop All Memo" )
      Coil( "RGHT Allowed Memo" )
   END_RUNG
   RUNG wire#powerrail
      Contact( "RGHT Allowed Memo" )
      wire#w1
      Contact( "RGHT L1 Memo" )
      wire#w2
      Move(in := "Speed L1 Memo", out1 => "Left Driver Analog input")
   END_RUNG
   RUNG wire#w2
      Move(in := "Speed L1 Memo", out1 => "Right Driver Analog input")
   END_RUNG
   RUNG wire#w1
      Contact( "RGHT L2 Memo" )
      wire#w3
      Move(in := "Speed L2 Memo", out1 => "Left Driver Analog input")
   END_RUNG
   RUNG wire#w3
      Move(in := "Speed L2 Memo", out1 => "Right Driver Analog input")
   END_RUNG
   RUNG wire#w1
      Contact( "RGHT L3 Memo" )
      wire#w4
      Move(in := "Speed L3 Memo", out1 => "Left Driver Analog input")
   END_RUNG
   RUNG wire#w4
      Move(in := "Speed L3 Memo", out1 => "Right Driver Analog input")
   END_RUNG
   RUNG wire#w1
      Contact( "RGHT L1 Memo" )
      wire#w5
      Coil( "Right G120C Stop Memo" )
   END_RUNG
   RUNG wire#w1
      Contact( "RGHT L2 Memo" )
   END_RUNG wire#w5
   RUNG wire#w1
      Contact( "RGHT L3 Memo" )
   END_RUNG wire#w5
   // the same network as SCL:
   "RGHT Allowed Memo" := "OK Memo" AND NOT "Cross M Memo" AND NOT "RGHT Stop All Memo";
   IF "RGHT Allowed Memo" AND "RGHT L1 Memo" THEN
       "Left Driver Analog input" := "Speed L1 Memo";
       "Right Driver Analog input" := "Speed L1 Memo";
   END_IF;
   IF "RGHT Allowed Memo" AND "RGHT L2 Memo" THEN
       "Left Driver Analog input" := "Speed L2 Memo";
       "Right Driver Analog input" := "Speed L2 Memo";
   END_IF;
   IF "RGHT Allowed Memo" AND "RGHT L3 Memo" THEN
       "Left Driver Analog input" := "Speed L3 Memo";
       "Right Driver Analog input" := "Speed L3 Memo";
   END_IF;
   "Right G120C Stop Memo" := "RGHT Allowed Memo" AND ("RGHT L1 Memo" OR "RGHT L2 Memo" OR "RGHT L3 Memo");
END_REGION

REGION Network 15: Tunnel FW-LFT
   RUNG wire#powerrail
      Contact( "OK Memo" )
      Contact( "Cross M Memo" )
      I_Contact( "FW Stop All Memo" )
      I_Contact( "LFT Stop All Memo" )
      Coil( "FW-LFT Allowed Memo" )
   END_RUNG
   RUNG wire#powerrail
      Contact( "FW-LFT Allowed Memo" )
      Contact( "FW-LFT Memo" )
      wire#w1
      Move(in := "Speed L2 Memo", out1 => "Right Driver Analog input")
   END_RUNG
   RUNG wire#w1
      { S7_Templates := "SrcType := Int" } Mul(in1 := "Speed L2 Memo", in2 := 2, out => "Left Driver Analog input")
   END_RUNG
   RUNG wire#w1
      Contact( "FW-LFT Memo" )
      Coil( "FW-LFT G120C Stop Memo" )
   END_RUNG
   // the same network as SCL:
   "FW-LFT Allowed Memo" := "OK Memo" AND "Cross M Memo" AND NOT "FW Stop All Memo" AND NOT "LFT Stop All Memo";
   #_w1 := "FW-LFT Allowed Memo" AND "FW-LFT Memo";
   IF #_w1 THEN
       "Right Driver Analog input" := "Speed L2 Memo";
       "Left Driver Analog input" := "Speed L2 Memo" * 2;
   END_IF;
   "FW-LFT G120C Stop Memo" := #_w1 AND "FW-LFT Memo";
END_REGION

REGION Network 16: Tunnel FW-RGHT
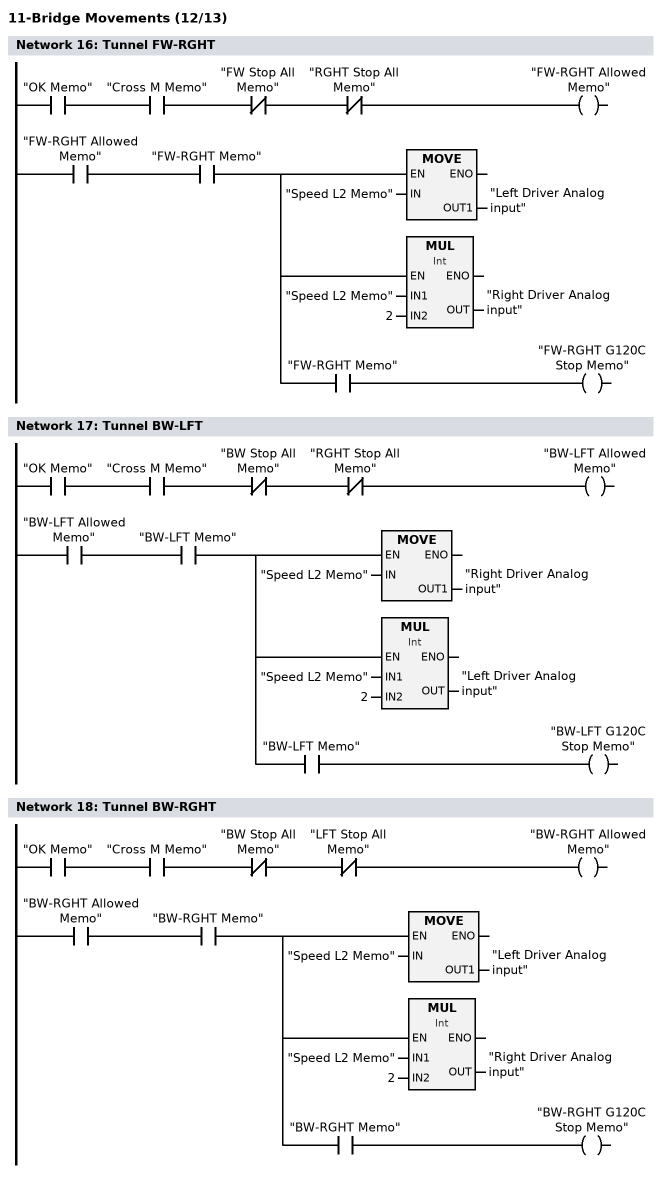
   RUNG wire#powerrail
      Contact( "OK Memo" )
      Contact( "Cross M Memo" )
      I_Contact( "FW Stop All Memo" )
      I_Contact( "RGHT Stop All Memo" )
      Coil( "FW-RGHT Allowed Memo" )
   END_RUNG
   RUNG wire#powerrail
      Contact( "FW-RGHT Allowed Memo" )
      Contact( "FW-RGHT Memo" )
      wire#w1
      Move(in := "Speed L2 Memo", out1 => "Left Driver Analog input")
   END_RUNG
   RUNG wire#w1
      { S7_Templates := "SrcType := Int" } Mul(in1 := "Speed L2 Memo", in2 := 2, out => "Right Driver Analog input")
   END_RUNG
   RUNG wire#w1
      Contact( "FW-RGHT Memo" )
      Coil( "FW-RGHT G120C Stop Memo" )
   END_RUNG
   // the same network as SCL:
   "FW-RGHT Allowed Memo" := "OK Memo" AND "Cross M Memo" AND NOT "FW Stop All Memo" AND NOT "RGHT Stop All Memo";
   #_w1 := "FW-RGHT Allowed Memo" AND "FW-RGHT Memo";
   IF #_w1 THEN
       "Left Driver Analog input" := "Speed L2 Memo";
       "Right Driver Analog input" := "Speed L2 Memo" * 2;
   END_IF;
   "FW-RGHT G120C Stop Memo" := #_w1 AND "FW-RGHT Memo";
END_REGION

REGION Network 17: Tunnel BW-LFT
   RUNG wire#powerrail
      Contact( "OK Memo" )
      Contact( "Cross M Memo" )
      I_Contact( "BW Stop All Memo" )
      I_Contact( "RGHT Stop All Memo" )
      Coil( "BW-LFT Allowed Memo" )
   END_RUNG
   RUNG wire#powerrail
      Contact( "BW-LFT Allowed Memo" )
      Contact( "BW-LFT Memo" )
      wire#w1
      Move(in := "Speed L2 Memo", out1 => "Right Driver Analog input")
   END_RUNG
   RUNG wire#w1
      { S7_Templates := "SrcType := Int" } Mul(in1 := "Speed L2 Memo", in2 := 2, out => "Left Driver Analog input")
   END_RUNG
   RUNG wire#w1
      Contact( "BW-LFT Memo" )
      Coil( "BW-LFT G120C Stop Memo" )
   END_RUNG
   // the same network as SCL:
   "BW-LFT Allowed Memo" := "OK Memo" AND "Cross M Memo" AND NOT "BW Stop All Memo" AND NOT "RGHT Stop All Memo";
   #_w1 := "BW-LFT Allowed Memo" AND "BW-LFT Memo";
   IF #_w1 THEN
       "Right Driver Analog input" := "Speed L2 Memo";
       "Left Driver Analog input" := "Speed L2 Memo" * 2;
   END_IF;
   "BW-LFT G120C Stop Memo" := #_w1 AND "BW-LFT Memo";
END_REGION

REGION Network 18: Tunnel BW-RGHT
   RUNG wire#powerrail
      Contact( "OK Memo" )
      Contact( "Cross M Memo" )
      I_Contact( "BW Stop All Memo" )
      I_Contact( "LFT Stop All Memo" )
      Coil( "BW-RGHT Allowed Memo" )
   END_RUNG
   RUNG wire#powerrail
      Contact( "BW-RGHT Allowed Memo" )
      Contact( "BW-RGHT Memo" )
      wire#w1
      Move(in := "Speed L2 Memo", out1 => "Left Driver Analog input")
   END_RUNG
   RUNG wire#w1
      { S7_Templates := "SrcType := Int" } Mul(in1 := "Speed L2 Memo", in2 := 2, out => "Right Driver Analog input")
   END_RUNG
   RUNG wire#w1
      Contact( "BW-RGHT Memo" )
      Coil( "BW-RGHT G120C Stop Memo" )
   END_RUNG
   // the same network as SCL:
   "BW-RGHT Allowed Memo" := "OK Memo" AND "Cross M Memo" AND NOT "BW Stop All Memo" AND NOT "LFT Stop All Memo";
   #_w1 := "BW-RGHT Allowed Memo" AND "BW-RGHT Memo";
   IF #_w1 THEN
       "Left Driver Analog input" := "Speed L2 Memo";
       "Right Driver Analog input" := "Speed L2 Memo" * 2;
   END_IF;
   "BW-RGHT G120C Stop Memo" := #_w1 AND "BW-RGHT Memo";
END_REGION

REGION Network 19: Drivers ON & Reversing !!!!
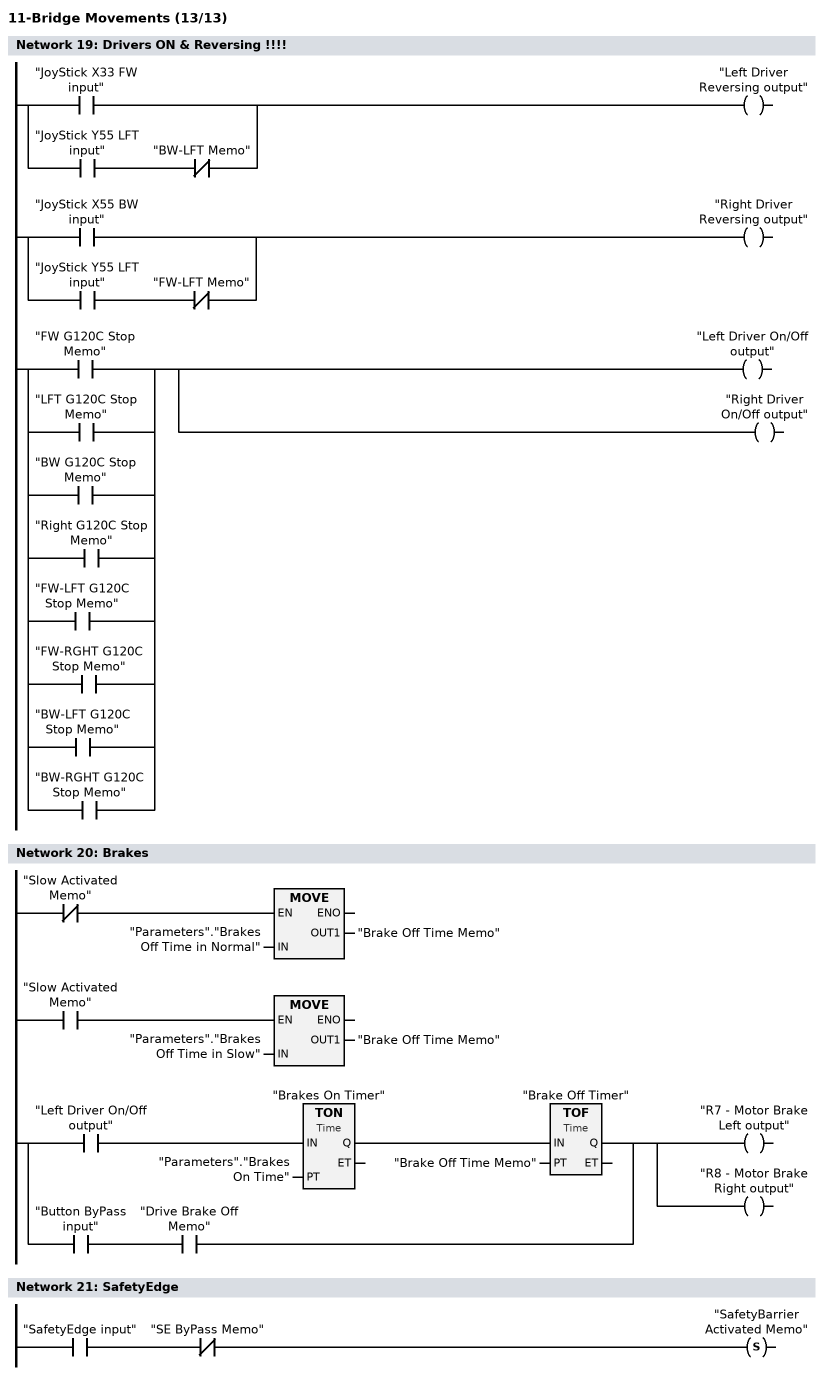
   RUNG wire#powerrail
      Contact( "JoyStick X33 FW input" )
      wire#w1
      Coil( "Left Driver Reversing output" )
   END_RUNG
   RUNG wire#powerrail
      Contact( "JoyStick Y55 LFT input" )
      I_Contact( "BW-LFT Memo" )
   END_RUNG wire#w1
   RUNG wire#powerrail
      Contact( "JoyStick X55 BW input" )
      wire#w2
      Coil( "Right Driver Reversing output" )
   END_RUNG
   RUNG wire#powerrail
      Contact( "JoyStick Y55 LFT input" )
      I_Contact( "FW-LFT Memo" )
   END_RUNG wire#w2
   RUNG wire#powerrail
      Contact( "FW G120C Stop Memo" )
      wire#w3
      Coil( "Left Driver On/Off output" )
   END_RUNG
   RUNG wire#powerrail
      Contact( "LFT G120C Stop Memo" )
   END_RUNG wire#w3
   RUNG wire#powerrail
      Contact( "BW G120C Stop Memo" )
   END_RUNG wire#w3
   RUNG wire#powerrail
      Contact( "Right G120C Stop Memo" )
   END_RUNG wire#w3
   RUNG wire#powerrail
      Contact( "FW-LFT G120C Stop Memo" )
   END_RUNG wire#w3
   RUNG wire#powerrail
      Contact( "FW-RGHT G120C Stop Memo" )
   END_RUNG wire#w3
   RUNG wire#powerrail
      Contact( "BW-LFT G120C Stop Memo" )
   END_RUNG wire#w3
   RUNG wire#powerrail
      Contact( "BW-RGHT G120C Stop Memo" )
   END_RUNG wire#w3
   RUNG wire#w3
      Coil( "Right Driver On/Off output" )
   END_RUNG
   // the same network as SCL:
   "Left Driver Reversing output" := "JoyStick X33 FW input" OR ("JoyStick Y55 LFT input" AND NOT "BW-LFT Memo");
   "Right Driver Reversing output" := "JoyStick X55 BW input" OR ("JoyStick Y55 LFT input" AND NOT "FW-LFT Memo");
   "Left Driver On/Off output" := "FW G120C Stop Memo" OR "LFT G120C Stop Memo" OR "BW G120C Stop Memo" OR "Right G120C Stop Memo" OR "FW-LFT G120C Stop Memo" OR "FW-RGHT G120C Stop Memo" OR "BW-LFT G120C Stop Memo" OR "BW-RGHT G120C Stop Memo";
   "Right Driver On/Off output" := "Left Driver On/Off output";
END_REGION

REGION Network 20: Brakes
   RUNG wire#powerrail
      I_Contact( "Slow Activated Memo" )
      Move(in := "Parameters"."Brakes Off Time in Normal", out1 => "Brake Off Time Memo")
   END_RUNG
   RUNG wire#powerrail
      Contact( "Slow Activated Memo" )
      Move(in := "Parameters"."Brakes Off Time in Slow", out1 => "Brake Off Time Memo")
   END_RUNG
   RUNG wire#powerrail
      Contact( "Left Driver On/Off output" )
      { S7_Templates := "time_type := Time" } "Brakes On Timer".TON(pt := "Parameters"."Brakes On Time", et =>)
      { S7_Templates := "time_type := Time" } "Brake Off Timer".TOF(pt := "Brake Off Time Memo", et =>)
      wire#w1
      Coil( "R7 - Motor Brake Left output" )
   END_RUNG
   RUNG wire#powerrail
      Contact( "Button ByPass input" )
      Contact( "Drive Brake Off Memo" )
   END_RUNG wire#w1
   RUNG wire#w1
      Coil( "R8 - Motor Brake Right output" )
   END_RUNG
   // the same network as SCL:
   IF NOT "Slow Activated Memo" THEN
       "Brake Off Time Memo" := "Parameters"."Brakes Off Time in Normal";
   END_IF;
   IF "Slow Activated Memo" THEN "Brake Off Time Memo" := "Parameters"."Brakes Off Time in Slow"; END_IF;
   "Brakes On Timer".TON(IN := "Left Driver On/Off output", PT := "Parameters"."Brakes On Time");
   "Brake Off Timer".TOF(IN := "Brakes On Timer".Q, PT := "Brake Off Time Memo");
   "R7 - Motor Brake Left output" := "Brake Off Timer".Q OR ("Button ByPass input" AND "Drive Brake Off Memo");
   "R8 - Motor Brake Right output" := "R7 - Motor Brake Left output";
END_REGION

REGION Network 21: SafetyEdge
   RUNG wire#powerrail
      Contact( "SafetyEdge input" )
      I_Contact( "SE ByPass Memo" )
      S_Coil( "SafetyBarrier Activated Memo" )
   END_RUNG
   // the same network as SCL:
   IF "SafetyEdge input" AND NOT "SE ByPass Memo" THEN "SafetyBarrier Activated Memo" := TRUE; END_IF;
END_REGION
END_ORGANIZATION_BLOCK
